# EPICS substitutions: exampleApp/example/exampleApp/Db/user.substitutions
# Example substitutions file

file "db/dbExample1.db" {
    { user = "yifans" }
}

file db/dbExample2.db {
    pattern { user, no, scan }
        { "yifans", 1, "1 second" }
        { "yifans", 2, "2 second" }
        { "yifans", 3, "5 second" }
}
